// TIA Portal project "ISA_P12" (V16)

(* hardware
DEVICE "S7-1200 station_1"  S7-1200 Station
   slot 0: "Rack_0"  S7-1200 Rack  Rack  V1.0
   slot 1: "PLC_1"  CPU 1215C DC/DC/DC  6ES7 215-1AG40-0XB0  V4.4
DEVICE "SINAMICS G_1"  Sinamics.Device
   slot 0: "	_0"  Rail  SinamicsG120CRackP
   slot 0: "Accionamiento_1"  G120C PN  6SL3210-1KE11-8UF1  4.7
      slot 1: "Interfaz PROFINET"  MDD-SinamicsG120-P
      slot 3: "PM G120C"  PM G120C  6SL3210-1KE11-8UF1  -
DEVICE "PC-System_1"  SIMATIC PC station
   slot 0: "Estación PC SIMATIC"  Rail  SIMATIC PC-Station  V1.0
      slot 125: "Stationmanager"  Station_Manager  V6.0.4
   slot 1: "HMI_RT_1"  WinCC RT Advanced  6AV2 104-0xxxx-xxxx  16.0.0.0
      slot 33792: "Interfaz del equipo"  Host interface
   slot 2: "IE general_1"  IE General  IE_CP  V8.2.0
*)

// ===== PLC "PLC_1"  CPU 1215C DC/DC/DC =====

VAR_GLOBAL   // PLC tag table "Tabla de variables estándar"
   "recibir_variador" AT %QW256 : Word;
   "consigna_principal" AT %QW258 : Word;
   "servicio_habilitado" AT %I256.2 : Bool;
   "velocidad_maxima_alcanzada" AT %I257.2 : Bool;
   "velocidad_real" AT %IW258 : Word;
   "enviar_variador" AT %IW256 : Word;
   "Tag_1" AT %M10.0 : Bool;
   "Eje_1_Drive_IN" AT %I256.0 : "PD_TEL1_IN";
   "Eje_1_Drive_OUT" AT %Q256.0 : "PD_TEL1_OUT";
   "HSC_1_A" AT %I0.0 : Bool;
   "HSC_1_B" AT %I0.1 : Bool;
   "Eje_1_PassiveHomingSwitch" AT %I0.2 : Bool;
   "Clock_Byte" AT %MB0 : Byte;
   "Clock_10Hz" AT %M0.0 : Bool;
   "Clock_5Hz" AT %M0.1 : Bool;
   "Clock_2.5Hz" AT %M0.2 : Bool;
   "Clock_2Hz" AT %M0.3 : Bool;
   "Clock_1.25Hz" AT %M0.4 : Bool;
   "Clock_1Hz" AT %M0.5 : Bool;
   "Clock_0.625Hz" AT %M0.6 : Bool;
   "Clock_0.5Hz" AT %M0.7 : Bool;
   "System_Byte" AT %MB1 : Byte;
   "FirstScan" AT %M1.0 : Bool;
   "DiagStatusUpdate" AT %M1.1 : Bool;
   "AlwaysTRUE" AT %M1.2 : Bool;
   "AlwaysFALSE" AT %M1.3 : Bool;
END_VAR

DATA_BLOCK "Variables"   // DB1
{ S7_Optimized_Access := 'TRUE' }
VERSION : 0.1
   VAR
      power_scada : Bool;
      stop_scada : Bool;
      home_scada : Bool;
      modo_scada : Int;
      reset_scada : Bool;
      move_velocity_scada : Bool;
      move_relative_scada : Bool;
      move_absolute_scada : Bool;
      velocidad_velocity_scada : Real;
      distancia_relative_scada : Real;
      velocidad_relative_scada : Real;
      posicion_absolute_scada : Real;
      velocidad_absolute_scada : Real;
      posicion_actual_scada : Real;
      velocidad_actual_scada : Real;
      posicion_scada : Real;
      velocidad_scada : Real;
      medir_scada : Bool;
      medida_mm : Real;
      home_medida : Bool;
      etapa : Int;
      posicion_inicial : Real;
      posicion_final : Real;
   END_VAR
BEGIN
END_DATA_BLOCK

DATA_BLOCK "Eje_1"   // DB5, Motion_DB
{ S7_Optimized_Access := 'TRUE' }
AUTHOR : SIMATIC
FAMILY : BasicMC
NAME : TO_PosAx
VERSION : 7.0
// stored: InstanceOfName TO_PositioningAxis
"TO_PositioningAxis"
BEGIN
   // Axis.LengthUnitNormalized.Time = 1
   // Axis.HomingReferencePointSwitch_AddressCU = %I0.2
   // Axis.PassiveHomingReferencePointSwitch_AddressCU = %I0.2
   // Axis.Encoder.OperatingPhaseCU = 2
   // Axis.Encoder.SelectedClockGenerator2EnumCU = %I0.1
   // Axis.Encoder.SelectedClockGenerator1EnumCU = %I0.0
   // Axis.Drive.OfflineDataAdaption = TRUE
   // Axis.Drive.TelegramAddressOutCU = %Q256.0
   // Axis.Drive.TelegramAddressInCU = %I256.0
   // Axis.Drive.DoNameCU = Accionamiento_1.Telegrama_estándar_1
   // Axis.LengthUnitNormalized.Distance = -2
   // Axis.Encoder.DbTypeCU = Classic
   // Axis.Drive.DbTypeCU = Classic
END_DATA_BLOCK

ORGANIZATION_BLOCK "Main"   // OB1, LAD, ProgramCycle
TITLE = "Main Program Sweep (Cycle)"
{ S7_Optimized_Access := 'TRUE' }
VERSION : 0.1
   VAR_INPUT
      Initial_Call : Bool;   // Initial call of this OB
      Remanence : Bool;   // =True, if remanent data are available
   END_VAR
BEGIN

REGION Network 1: Power
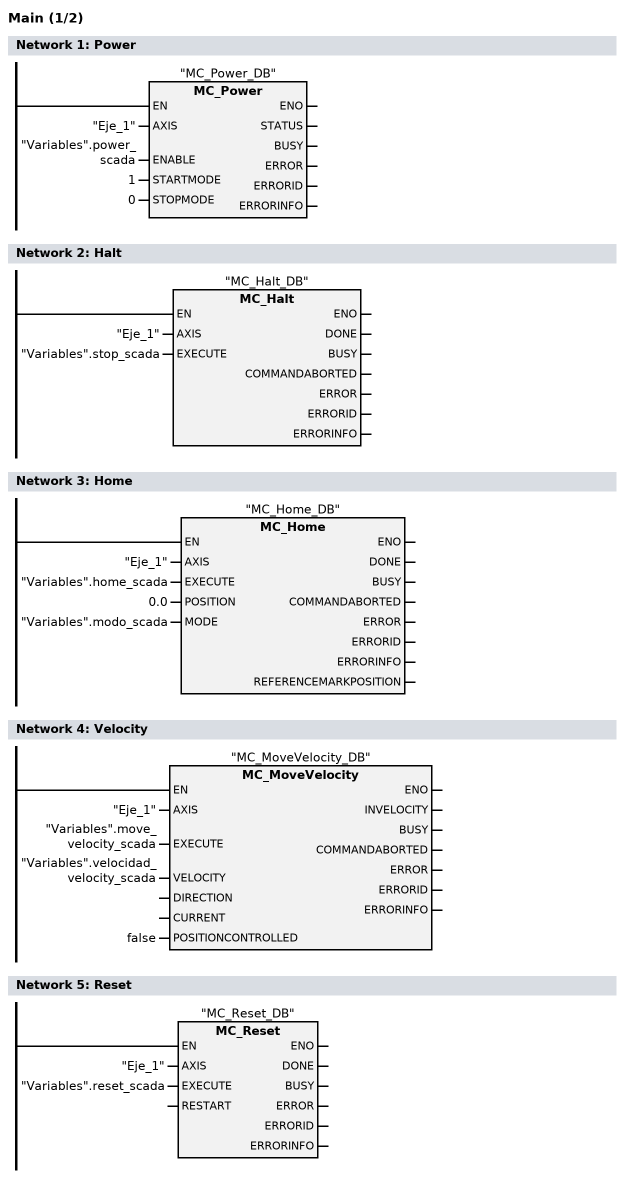
   "MC_Power_DB"(Axis := "Eje_1", Enable := "Variables".power_scada, StartMode := 1, StopMode := 0);   // MC_Power
END_REGION

REGION Network 2: Halt
   "MC_Halt_DB"(Axis := "Eje_1", Execute := "Variables".stop_scada);   // MC_Halt
END_REGION

REGION Network 3: Home
   "MC_Home_DB"(Axis := "Eje_1",   // MC_Home
                Execute := "Variables".home_scada,
                Position := 0.0,
                Mode := "Variables".modo_scada);
END_REGION

REGION Network 4: Velocity
   "MC_MoveVelocity_DB"(Axis := "Eje_1",   // MC_MoveVelocity
                        Execute := "Variables".move_velocity_scada,
                        Velocity := "Variables".velocidad_velocity_scada,
                        PositionControlled := false);
END_REGION

REGION Network 5: Reset
   "MC_Reset_DB"(Axis := "Eje_1", Execute := "Variables".reset_scada);   // MC_Reset
END_REGION

REGION Network 6: Relative
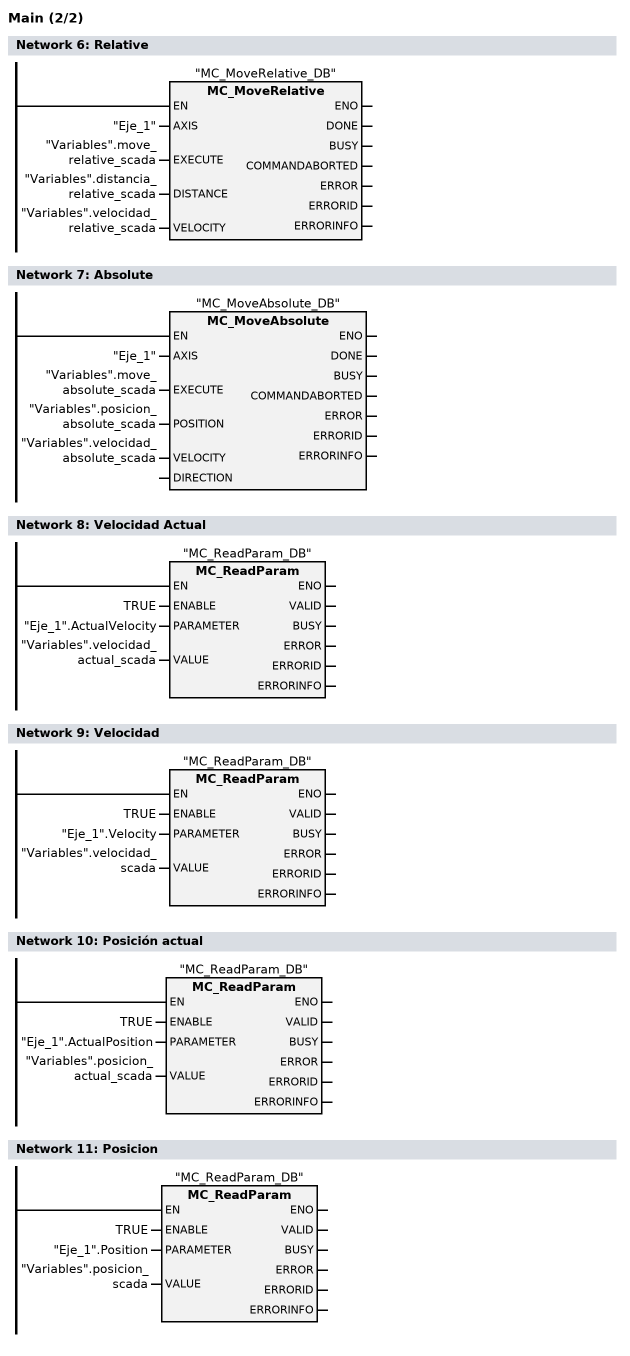
   "MC_MoveRelative_DB"(Axis := "Eje_1",   // MC_MoveRelative
                        Execute := "Variables".move_relative_scada,
                        Distance := "Variables".distancia_relative_scada,
                        Velocity := "Variables".velocidad_relative_scada);
END_REGION

REGION Network 7: Absolute
   "MC_MoveAbsolute_DB"(Axis := "Eje_1",   // MC_MoveAbsolute
                        Execute := "Variables".move_absolute_scada,
                        Position := "Variables".posicion_absolute_scada,
                        Velocity := "Variables".velocidad_absolute_scada);
END_REGION

REGION Network 8: Velocidad Actual
   "MC_ReadParam_DB"(Enable := TRUE,   // MC_ReadParam
                     Parameter := "Eje_1".ActualVelocity,
                     Value := "Variables".velocidad_actual_scada);
END_REGION

REGION Network 9: Velocidad
   "MC_ReadParam_DB"(Enable := TRUE, Parameter := "Eje_1".Velocity, Value := "Variables".velocidad_scada);   // MC_ReadParam
END_REGION

REGION Network 10: Posición actual
   "MC_ReadParam_DB"(Enable := TRUE,   // MC_ReadParam
                     Parameter := "Eje_1".ActualPosition,
                     Value := "Variables".posicion_actual_scada);
END_REGION

REGION Network 11: Posicion
   "MC_ReadParam_DB"(Enable := TRUE, Parameter := "Eje_1".Position, Value := "Variables".posicion_scada);   // MC_ReadParam
END_REGION
END_ORGANIZATION_BLOCK

ORGANIZATION_BLOCK "medir_pieza"   // OB123, LAD, ProgramCycle
TITLE = "Main Program Sweep (Cycle)"
{ S7_Optimized_Access := 'TRUE' }
VERSION : 0.1
   VAR_INPUT
      Initial_Call : Bool;   // Initial call of this OB
      Remanence : Bool;   // =True, if remanent data are available
   END_VAR
   VAR_TEMP
      midiendo : Bool;
      move_medir : Bool;
      retroceder : Bool;
      retroceder_done : Bool;
      tiempo : Real;
      inicio : Bool;
      etapa : Int;
      move_zero : Bool;
      posicion_inicial : Real;
      posicion_final : Real;
      velocity : Real;
      medida : Real;
   END_VAR
BEGIN

REGION Network 1 (SCL)
   IF "FirstScan" THEN
       "Variables".etapa := 0;
   END_IF;

   CASE "Variables".etapa OF
       0:
           IF "Variables".medir_scada THEN
               "Variables".etapa := 1;
           END_IF;
       1:
           #velocity := 50.0;
           #move_medir := TRUE;
           IF "Eje_1_PassiveHomingSwitch" THEN
               "Variables".posicion_inicial := "Variables".posicion_actual_scada;
               "Variables".etapa := 2;
           END_IF;
       2:
           IF NOT "Eje_1_PassiveHomingSwitch" THEN
               "Variables".posicion_final := "Variables".posicion_actual_scada;
               "Variables".etapa := 3;
           END_IF;
       3:
           "Variables".medida_mm := "Variables".posicion_final - "Variables".posicion_inicial;
           #velocity := 0.0;
           #move_medir := TRUE;
           "Variables".etapa := 0;
   END_CASE;
END_REGION

REGION Network 2
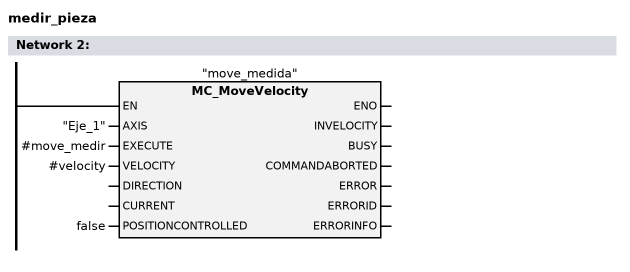
   "move_medida"(Axis := "Eje_1", Execute := #move_medir, Velocity := #velocity, PositionControlled := false);   // MC_MoveVelocity
END_REGION
END_ORGANIZATION_BLOCK

(* ===== HMI "HMI_RT_1" =====
system functions are stored by id; their names below are inferred from use
connection "HMI_Conexión_1": ETHERNET, S7_1200_OMS

HMI tags "Tabla de variables estándar"
   "Variables_stop_scada" : Bool = PLC Variables.stop_scada, 1 s
   "Variables_power_scada" : Bool = PLC Variables.power_scada, 1 s
   "Variables_home_scada" : Bool = PLC Variables.home_scada, 1 s
   "Variables_modo_scada" : Int = PLC Variables.modo_scada, 1 s
   "Variables_reset_scada" : Bool = PLC Variables.reset_scada, 1 s
   "Variables_move_velocity_scada" : Bool = PLC Variables.move_velocity_scada, 1 s
   "Variables_move_relative_scada" : Bool = PLC Variables.move_relative_scada, 1 s
   "Variables_move_absolute_scada" : Bool = PLC Variables.move_absolute_scada, 1 s
   "Variables_velocidad_velocity_scada" : Real = PLC Variables.velocidad_velocity_scada, 1 s
   "Variables_distancia_relative_scada" : Real = PLC Variables.distancia_relative_scada, 1 s
   "Variables_velocidad_relative_scada" : Real = PLC Variables.velocidad_relative_scada, 1 s
   "Variables_posicion_absolute_scada" : Real = PLC Variables.posicion_absolute_scada, 1 s
   "Variables_velocidad_absolute_scada" : Real = PLC Variables.velocidad_absolute_scada, 1 s
   "Variables_posicion_actual_scada" : Real = PLC Variables.posicion_actual_scada, 100 ms
   "Variables_posicion_scada" : Real = PLC Variables.posicion_scada, 100 ms
   "Variables_velocidad_actual_scada" : Real = PLC Variables.velocidad_actual_scada, 100 ms
   "Variables_velocidad_scada" : Real = PLC Variables.velocidad_scada, 100 ms
   "Variables_medida_mm" : Real = PLC Variables.medida_mm, 1 s
   "Variables_medir_scada" : Bool = PLC Variables.medir_scada, 1 s

screen "Imagen_1" 800x600
   Switch "Interruptor_1" at 51,42 size 150x82; CaptionText 'Power'; TextOff 'OFF'; TextOn 'ON'
      ProcessValue <- "Variables_power_scada"
   Button "Botón_1" at 51,165 size 151x67; TextOff 'STOP'
      on Press: SetBit("Variables_stop_scada")
      on Release: ResetBit("Variables_stop_scada")
   IOField "Campo ES_1" at 116,442 size 84x37; FormatPattern 9
      ProcessValue <- "Variables_modo_scada"
   TextField "Campo de texto_1" at 56,444 size 58x27; Text 'Modo'
   Button "Botón_2" at 44,514 size 150x40; TextOff 'RESET'
      on Press: SetBit("Variables_reset_scada")
      on Release: ResetBit("Variables_reset_scada")
   Button "Botón_3" at 294,38 size 147x64; TextOff 'MOVE Velocity'
      on Press: SetBit("Variables_move_velocity_scada")
      on Release: ResetBit("Variables_move_velocity_scada")
   Button "Botón_4" at 295,118 size 146x64; TextOff 'MOVE Relative'
      on Press: SetBit("Variables_move_relative_scada")
      on Release: ResetBit("Variables_move_relative_scada")
   Button "Botón_5" at 295,199 size 146x65; TextOff 'MOVE Absolute'
      on Press: SetBit("Variables_move_absolute_scada")
      on Release: ResetBit("Variables_move_absolute_scada")
   IOField "Campo ES_2" at 457,59 size 114x38; FormatPattern 999.9
      ProcessValue <- "Variables_velocidad_velocity_scada"
   TextField "Campo de texto_2" at 468,111 size 93x27; Text 'Distancia'
   TextField "Campo de texto_3" at 463,31 size 98x27; Text 'Velocidad'
   TextField "Campo de texto_4" at 624,197 size 98x27; Text 'Velocidad'
   TextField "Campo de texto_5" at 472,196 size 85x27; Text 'Posición'
   TextField "Campo de texto_10" at 51,277 size 64x27; Text 'HOME'
   IOField "Campo ES_3" at 457,136 size 115x38; FormatPattern s999.9
      ProcessValue <- "Variables_distancia_relative_scada"
   IOField "Campo ES_4" at 457,222 size 114x38; FormatPattern s999.9
      ProcessValue <- "Variables_posicion_absolute_scada"
   IOField "Campo ES_5" at 617,136 size 119x38; FormatPattern s999.9
      ProcessValue <- "Variables_velocidad_relative_scada"
   IOField "Campo ES_6" at 618,222 size 118x38; FormatPattern s999.9
      ProcessValue <- "Variables_velocidad_absolute_scada"
   TextField "Campo de texto_6" at 325,315 size 151x27; Text 'Posición Actual'
   IOField "Campo ES_7" at 318,340 size 169x38; FormatPattern s999.99
      ProcessValue <- "Variables_posicion_actual_scada"
   TextField "Campo de texto_7" at 353,391 size 85x27; Text 'Posición'
   IOField "Campo ES_8" at 318,419 size 169x38; FormatPattern s999.99
      ProcessValue <- "Variables_posicion_scada"
   TextField "Campo de texto_8" at 523,315 size 164x27; Text 'Velocidad Actual'
   IOField "Campo ES_9" at 521,340 size 169x38; FormatPattern 999.99
      ProcessValue <- "Variables_velocidad_actual_scada"
   TextField "Campo de texto_9" at 551,394 size 98x27; Text 'Velocidad'
   IOField "Campo ES_10" at 521,419 size 169x38; FormatPattern 999.99
      ProcessValue <- "Variables_velocidad_scada"
   Button "SB_NavigateHome_85x64_Mono" at 51,310 size 149x122; TextOff 'Text'; PictureOff "SB_NavigateHome_85x64_mono"
      on Press: SetBit("Variables_home_scada")
      on Release: ResetBit("Variables_home_scada")
   TextField "Campo de texto_11" at 624,109 size 98x27; Text 'Velocidad'
   Button "Botón_6" at 318,491 size 167x40; TextOff 'MEDIR'
      on Release: ResetBit("Variables_medir_scada")
      on Press: SetBit("Variables_medir_scada")
   IOField "Campo ES_11" at 523,491 size 169x40; FormatPattern 999.99; Unit mm
      ProcessValue <- "Variables_medida_mm"
*)